FUNCTION_BLOCK DoublePneumaticActuator EXTENDS PneumaticActuator

VAR
	extendOutput1 AT %Q* : BOOL;
	retractOutput1 AT %Q* : BOOL;
END_VAR

METHOD ExtendActuator : BOOL
extendOutput1 := TRUE;
retractOutput1 := FALSE;

SUPER^.ExtendActuator();
END_METHOD

METHOD RetractActuator : BOOL
RetractActuator := TRUE;
extendOutput := FALSE;
extendOutput1 := FALSE;
retractOutput := TRUE;
retractOutput1 := TRUE;

IF _logging THEN
	SendTraceData('Retracting...');
END_IF
END_METHOD

END_FUNCTION_BLOCK

(* stored: Version 1.1.0.1
   POU DoublePneumaticActuator: Id {350374c4-e35b-4588-a102-a9495299579d}, SpecialFunc None
   Method ExtendActuator: Id {5de02e6e-e492-4a69-ba79-315c2faa832a}
   Method RetractActuator: Id {98b13311-7620-436b-b04c-62f132a20bcb} *)
